FUNCTION_BLOCK AE2_DELAY (* Delayed event propagation (AE2 Adapter, bidirektional, 1 Event) *)
  (* Standard: 61499-2; Description: Copyright (c) 2026 HR Agrartechnik GmbH This program and the accompanying materials are made available under the terms of the Eclipse Public License 2.0 which is available at https://www.eclipse.org/legal/epl-2.0/ SPDX-License-Identifier: EPL-2.0 *)
  (* Version 1.0, 2026-09-17, Franz Höpfinger, HR Agrartechnik GmbH, Wrapper fuer E_DELAY ueber AE2-Adapter (bidirektional) - existierte im Projekt noch nicht (Franz: 'AE2_DELAY fehlt auch noch'), war faelschlich als bereits vorhanden angenommen worden. PT als ATM-Socket statt Klartext-InputVar, sauber initialisierbar ueber initval_ATM+INIT/INITO, analog zur selben Korrektur bei AE_DELAY/ASR2_DELAY. *)
  (* Version 1.1, 2026-09-17, Franz Höpfinger, HR Agrartechnik GmbH, Bugfix (4diac IDE Validation: 'Name: DT is a reserved keyword' - DT ist Abkuerzung fuer DATE_AND_TIME, IEC 61131-3-Keyword): Socket DT in PT (Preset Time, Standardname wie bei TON/TOF) umbenannt. *)
  (* Version 1.2, 2026-09-17, Franz Höpfinger, HR Agrartechnik GmbH, Bugfix (Franz: 'AE2_DELAY braucht 2 Zeiten, ein DELAY FORWARD und ein DELAY BACKWARD'): AE2 ist echt bidirektional (EI1/EO1 je Socket UND Plug) - bisher wurde nur die Vorwaerts-Richtung (IN.EO1->OUT.EO1) verzoegert. Jetzt 2 unabhaengige E_DELAY-Instanzen: Vorwaerts (IN.EO1->OUT.EO1, PT_FWD) und Rueckwaerts (OUT.EI1->IN.EI1, PT_BWD). *)
  (* Version 1.3, 2026-09-17, Franz Höpfinger, HR Agrartechnik GmbH, Bugfix (Franz: 'wenn AE_DELAY ein STOP hat, braucht auch AE2_DELAY ein STOP'): 2 zusaetzliche unidirektionale AE-Sockets STOP_FWD/STOP_BWD ergaenzt, je auf E_DELAY_FWD.STOP/E_DELAY_BWD.STOP verdrahtet - analog zu AE_DELAY.STOP, je Richtung getrennt stoppbar. *)
  PACKAGE adapter::events::bidirectional;
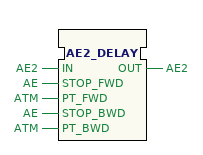
  SOCKETS
    IN : adapter::types::bidirectional::AE2; (* Event vom vorherigen Kettenglied (bidirektional: Vorwaerts herein, Rueckwaerts hinaus) *)
    STOP_FWD : adapter::types::unidirectional::AE; (* Stop delay Vorwaerts (analog AE_DELAY.STOP) *)
    PT_FWD : adapter::types::unidirectional::ATM; (* Preset Time Vorwaerts (IN->OUT), ATM statt Klartext-InputVar, sauber initialisierbar ueber initval_ATM *)
    STOP_BWD : adapter::types::unidirectional::AE; (* Stop delay Rueckwaerts *)
    PT_BWD : adapter::types::unidirectional::ATM; (* Preset Time Rueckwaerts (OUT->IN), unabhaengig von PT_FWD einstellbar *)
  END_SOCKETS
  PLUGS
    OUT : adapter::types::bidirectional::AE2; (* Verzoegertes Event, an naechstes Kettenglied (bidirektional: Vorwaerts hinaus, Rueckwaerts herein) *)
  END_PLUGS
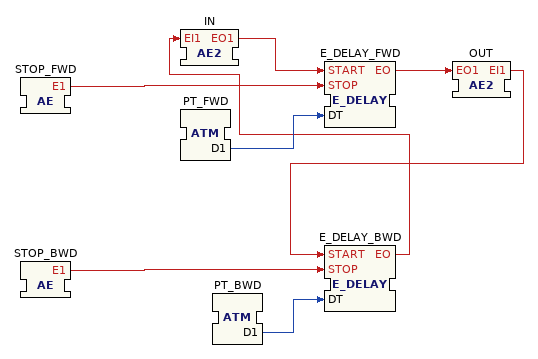
  FBS
    E_DELAY_FWD : iec61499::events::E_DELAY;
    E_DELAY_BWD : iec61499::events::E_DELAY;
  END_FBS
  EVENT_CONNECTIONS
    IN.EO1 TO E_DELAY_FWD.START;
    STOP_FWD.E1 TO E_DELAY_FWD.STOP;
    E_DELAY_FWD.EO TO OUT.EO1;
    OUT.EI1 TO E_DELAY_BWD.START;
    STOP_BWD.E1 TO E_DELAY_BWD.STOP;
    E_DELAY_BWD.EO TO IN.EI1;
  END_CONNECTIONS
  DATA_CONNECTIONS
    PT_FWD.D1 TO E_DELAY_FWD.DT;
    PT_BWD.D1 TO E_DELAY_BWD.DT;
  END_CONNECTIONS
END_FUNCTION_BLOCK
